TYPE XTSDiag_ModuleInfeedMapping_typ :
STRUCT
	Infeed		: INT;
	Position	: INT;
END_STRUCT
END_TYPE

(* stored: Version 1.1.0.1, ProductVersion 3.1.4026.12
   DUT XTSDiag_ModuleInfeedMapping_typ: Id {e89174bf-e0c3-0b0e-113d-82f7971572e1} *)
